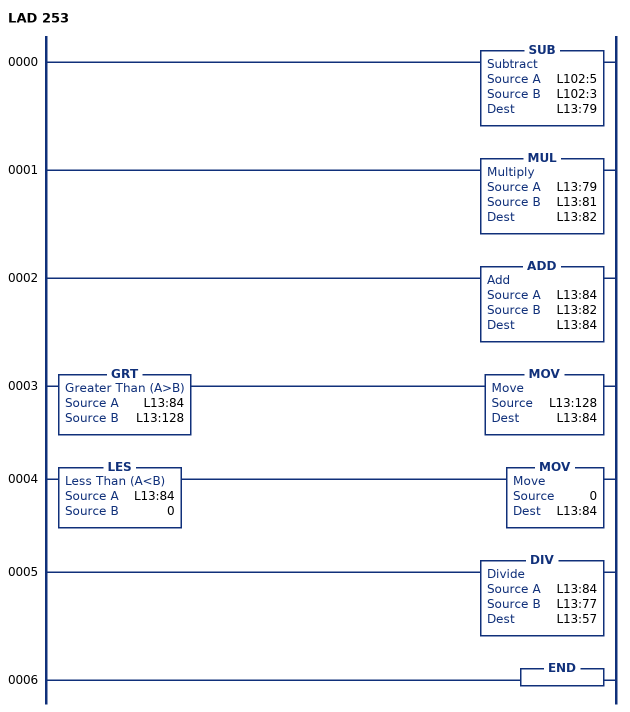
% Rung: 0 %
SOR SUB L102:5 L102:3 L13:79 EOR
% Rung: 1 %
SOR MUL L13:79 L13:81 L13:82 EOR
% Rung: 2 %
SOR ADD L13:84 L13:82 L13:84 EOR
% Rung: 3 %
SOR GRT L13:84 L13:128 MOV L13:128 L13:84 EOR
% Rung: 4 %
SOR LES L13:84 0 MOV 0 L13:84 EOR
% Rung: 5 %
SOR DIV L13:84 L13:77 L13:57 EOR
% Rung: 6 %
SOR END EOR

LADDER 254
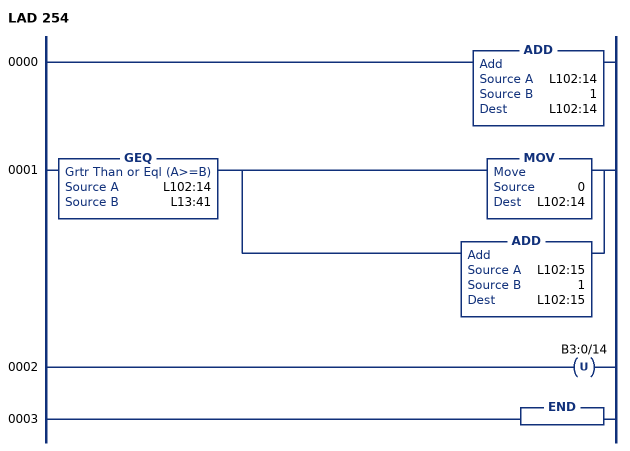
% Rung: 0 %
SOR ADD L102:14 1 L102:14 EOR
% Rung: 1 %
SOR GEQ L102:14 L13:41 BST MOV 0 L102:14 NXB ADD L102:15 1 L102:15 BND EOR
% Rung: 2 %
SOR OTU B3:0/14 EOR
% Rung: 3 %
SOR END EOR

LADDER 255
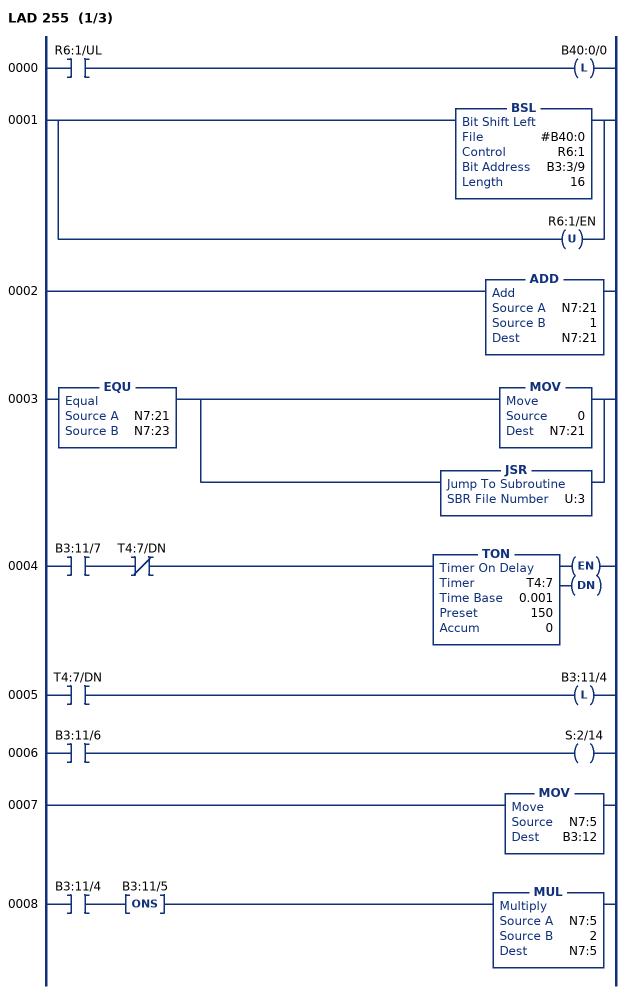
% Rung: 0 %
SOR XIC R6:1/UL OTL B40:0/0 EOR
% Rung: 1 %
SOR BST BSL #B40:0 R6:1 B3:3/9 16 NXB OTU R6:1/EN BND EOR
% Rung: 2 %
SOR ADD N7:21 1 N7:21 EOR
% Rung: 3 %
SOR EQU N7:21 N7:23 BST MOV 0 N7:21 NXB JSR U:3 BND EOR
% Rung: 4 %
SOR XIC B3:11/7 XIO T4:7/DN TON T4:7 0.001 150 0 EOR
% Rung: 5 %
SOR XIC T4:7/DN OTL B3:11/4 EOR
% Rung: 6 %
SOR XIC B3:11/6 OTE S:2/14 EOR
% Rung: 7 %
SOR MOV N7:5 B3:12 EOR
% Rung: 8 %
SOR XIC B3:11/4 ONS B3:11/5 MUL N7:5 2 N7:5 EOR

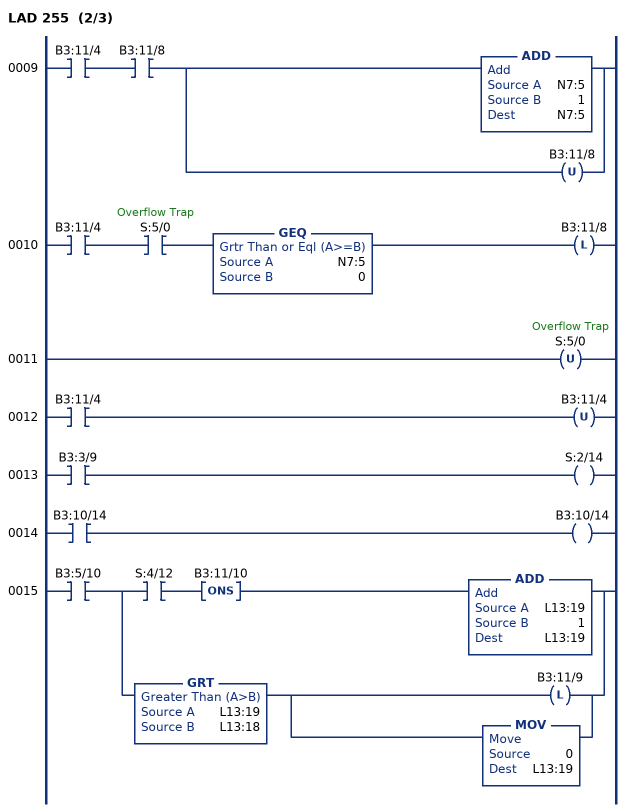
% Rung: 9 %
SOR XIC B3:11/4 XIC B3:11/8 BST ADD N7:5 1 N7:5 NXB OTU B3:11/8 BND EOR
% Rung: 10 %
SOR XIC B3:11/4 XIC S:5/0 GEQ N7:5 0 OTL B3:11/8 EOR
%   S:5/0  "Overflow Trap" %
% Rung: 11 %
SOR OTU S:5/0 EOR
%   S:5/0  "Overflow Trap" %
% Rung: 12 %
SOR XIC B3:11/4 OTU B3:11/4 EOR
% Rung: 13 %
SOR XIC B3:3/9 OTE S:2/14 EOR
% Rung: 14 %
SOR XIC B3:10/14 OTE B3:10/14 EOR
% Rung: 15 %
SOR XIC B3:5/10 BST XIC S:4/12 ONS B3:11/10 ADD L13:19 1 L13:19 NXB GRT L13:19 L13:18 BST OTL B3:11/9 NXB MOV 0 L13:19 BND BND EOR

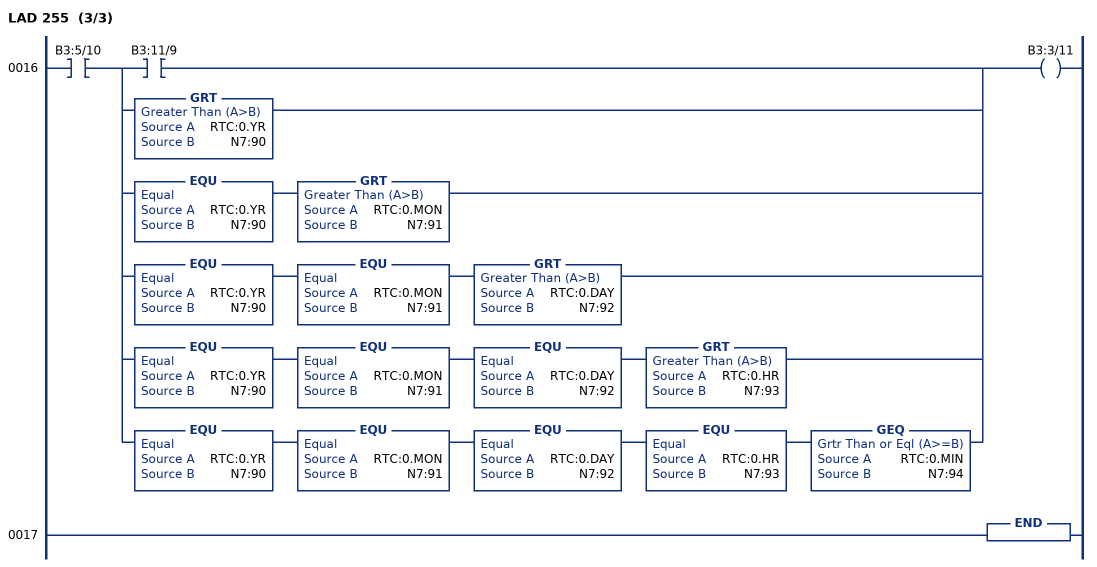
% Rung: 16 %
SOR XIC B3:5/10 BST XIC B3:11/9 NXB GRT RTC:0.YR N7:90 NXB EQU RTC:0.YR N7:90 GRT RTC:0.MON N7:91 NXB EQU RTC:0.YR N7:90 EQU RTC:0.MON N7:91 GRT RTC:0.DAY N7:92 NXB EQU RTC:0.YR N7:90 EQU RTC:0.MON N7:91 EQU RTC:0.DAY N7:92 GRT RTC:0.HR N7:93 NXB EQU RTC:0.YR N7:90 EQU RTC:0.MON N7:91 EQU RTC:0.DAY N7:92 EQU RTC:0.HR N7:93 GEQ RTC:0.MIN N7:94 BND OTE B3:3/11 EOR
% Rung: 17 %
SOR END EOR

DATA TABLE (non-zero values as saved)
DATA B3
% B3:0 % 0X88A2 0X0160 0X0001 0X5101 0X08A5 0X1540 0X0410 0X0461 0X5F80 0X2558
% B3:10 % 0X2000 0X40C7 0X4000 0X08D5 0X0000 0X0000 0X0000 0X0000 0X0000 0X0000
% B3:50 % 0X0001 0X0000 0X0000 0X0000 0X0000 0X0000 0X0000 0X0000 0X0000 0X0000
DATA T4
% .PRE .ACC %
% T4:0 % 0 1
% T4:1 % 150 0
% T4:2 % 400 0
% T4:3 % 222 61
% T4:4 % 1000 0
% T4:5 % 5 5
% T4:6 % 10 32766
% T4:7 % 150 0
% T4:8 % 20 13
% T4:9 % 50 44
% T4:10 % 200 0
% T4:11 % 111 0
% T4:12 % 40 96
% T4:13 % 250 0
% T4:14 % 666 0
% T4:15 % 1000 1006
% T4:16 % 400 0
% T4:17 % 100 96
% T4:18 % 5 0
% T4:19 % 300 0
% T4:20 % 200 0
% T4:21 % 200 0
% T4:22 % 200 0
% T4:23 % 250 0
% T4:24 % 666 0
% T4:25 % 666 0
% T4:26 % 666 0
% T4:27 % 250 0
% T4:28 % 250 0
% T4:29 % 5000 0
% T4:30 % 333 0
% T4:31 % 333 63
% T4:32 % 15 0
% T4:33 % 222 51
% T4:34 % 1111 0
DATA C5
% .PRE .ACC %
% C5:0 % 32766 0
DATA R6
% .LEN .POS %
% R6:0 % 1250 0
% R6:1 % 16 0
% R6:2 % 1050 0
% R6:3 % 1050 0
% R6:4 % 1250 0
% R6:5 % 1250 0
% R6:6 % 1713 0
% R6:7 % 16 0
% R6:8 % 1024 0
% R6:9 % 3 0
% R6:10 % 1713 0
% R6:11 % 1050 0
% R6:12 % 10 0
% R6:13 % 10 0
% R6:14 % 10 0
% R6:15 % 10 0
% R6:16 % 1713 0
% R6:17 % 1713 0
% R6:18 % 1050 0
% R6:19 % 10 0
DATA N7
% N7:0 % 32767 3 874 300 3 0 0 0 500 43
% N7:10 % 1000 43 0 8 8 8 1000 2000 50 1050
% N7:20 % 0 1329 16 2000 0 8 0 0 0 250
% N7:30 % 666 32767 150 0 728 1232 77 32 0 32
% N7:40 % 0 38 1 37 121 482 767 1350 16 0
% N7:50 % 0 0 0 16 1 900 0 0 32766 3
% N7:60 % 1713 1713 1050 871 1034 1024 4999 5 400 400
% N7:70 % 100 200 300 400 90 190 290 390 232 32767
% N7:80 % 0 0 1241 32767 1300 1310 61 26 10 1
% N7:90 % 2011 4 4 12 1 51 25 222 222 12
% N7:100 % 1003 90 110 100 175 25 0 0 0 0
% N7:190 % -128 27477 27605 32767 0 0 0 0 0 0
DATA F8
% F8:0 % 6
DATA L13
% L13:0 % 71471 190025 0 39179 291035
% L13:5 % 6415 33021 6415 172394 5190
% L13:10 % 5004 212369 41937 15 90
% L13:15 % 808527807 -2147483648 2147483647 2147483647 82058
% L13:20 % 147282566 -2001678473 777 36345 100
% L13:25 % 4777 7405 212365 0 713785867
% L13:30 % 94741822 6415 60000 -300674159 1444
% L13:35 % 0 5 99 1073770676 1073770698
% L13:40 % 0 1000000000 1000000 -291038042 -290955777
% L13:45 % 271741302 22 682 26 147282566
% L13:50 % 1099483545 682 1312162756 0 1099483625
% L13:55 % 283196 88766043 1774 47928606 47931497
% L13:60 % 7405 1860375 0 600 -1
% L13:65 % 100 -100 1088103355 -1153047802 1099483566
% L13:70 % 147282479 -1705050752 8 0 147282566
% L13:75 % 0 30 100 -392888222 5
% L13:80 % 40 74 370 40 177378
% L13:85 % 3144934 0 0 0 1099483588
% L13:90 % 283197 3 56648 5 -290955660
% L13:95 % 14 200235 0 271741575 10324515
% L13:100 % 400 7 2147483647 1111 1353
% L13:105 % 10324515 10670 147259324 212376 147259318
% L13:110 % 6 100 50 -2004823403 -2004823412
% L13:115 % -2004823407 5 3 -2004823410 26
% L13:120 % 87 212373 50 100 10
% L13:125 % 0 147282479 2147483647 3276500 3144930
% L13:130 % 2 2 0 99 0
% L13:135 % 0 0 3144930 5 70
% L13:140 % 0 5 36 50 50
% L13:145 % 683 5 88766044 5 0
% L13:150 % 12 20 4 -4 212369
% L13:155 % 0 -10 0 1 4589052
% L13:160 % 12573529 117 273 1220 45
% L13:165 % -2001679672 -2014253201 -2001679672 -2014253201 6706
% L13:170 % 12817 8 225 100 -2147483648
% L13:175 % 4 4 42 23 38
% L13:180 % 1088103355 0 0 1000000 0
% L13:185 % 0 0 -1153047802 0 0
DATA L19
% L19:0 % 713785867 713786507 713796116 713798249 713799019
% L19:5 % 713800070 713825116 713774048 713774596 713774802
% L19:10 % 713777491 713778421 713779204 713779851 713780015
% L19:15 % 713785499 713785672 0 0 0
DATA L20
% L20:0 % -290964835 -290964827 -290964819 -290964811 -290964803
% L20:5 % -290964795 -290964787 -290964779 -290964771 -290964763
% L20:10 % -290964755 -290964747 -290964739 -290964731 -290964723
% L20:15 % -290964715 -290964707 -290964699 -290964691 -290964683
% L20:20 % -290964675 -290964667 -290956009 -290956001 -290955993
% L20:25 % -290955985 -290955977 -290955969 -290955961 -290955953
% L20:30 % -290955945 -290955937 -290955929 -290955921 -290955913
% L20:35 % -290955905 -290955897 -290955889 -290955881 -290955873
% L20:40 % -290955865 -290955857 -290955849 -290955841 -290955833
% L20:45 % -290955825 -290955817 -290955809 -290955801 -290955793
% L20:50 % -290955785 -290955777 -290955769 -290955761 -290955753
% L20:55 % -290955745 -290955737 -290955729 -290955721 -290955713
% L20:60 % -290955705 -290955697 -290990460 -290986195 -290983780
% L20:65 % -290983772 -290983764 -290983756 -290983748 -290983740
% L20:70 % -290983732 -290983724 -290983716 -290981579 -290981571
% L20:75 % -290981563 -290981555 -290981547 -290981539 -290981531
% L20:80 % -290981523 -290981515 -290978966 -290978958 -290978950
% L20:85 % -290978942 -290978934 -290978926 -290978918 -290978910
% L20:90 % -290978902 -290964907 -290964899 -290964891 -290964883
% L20:95 % -290964875 -290964867 -290964859 -290964851 -290964843
DATA L21
% L21:0 % -2001679672 -2001679672 -2001679672 -2001679672 -2001679672
% L21:5 % -2001679672 -2001679672 -2001679672 -2001679672 -2001679672
% L21:10 % -2001679672 -2001679672 -2001679672 -2001679672 -2001679672
% L21:15 % -2001679672 -2001679672 -2001679672 -2001679672 -2001679672
% L21:20 % -2001679672 -2001679672 -2001679672 -2001679672 -2001679672
% L21:25 % -2001679672 -2001679672 -2001679672 -2001679672 -2001679672
% L21:30 % -2001679672 -2001679672 -2001679672 -2001679672 -2001679672
% L21:35 % -2001679672 -2001679672 -2001679672 -2001679672 -2001679672
% L21:40 % -2001679672 -2001679672 -2001679672 -2001679672 -2001679672
% L21:45 % -2001679672 -2001679672 -2001679672 -2001679672 -2001679672
% L21:50 % -2001679672 -2001679672 -2001679672 -2001679672 -2001679672
% L21:55 % -2001679672 -2001679672 -2001679672 -2001679672 -2001679672
% L21:60 % -2001679672 -2001679672 -2001679672 -2001679672 -2001679672
% L21:65 % -2001679672 -2001679672 -2001679672 -2001679672 -2001679672
% L21:70 % -2001679672 -2001679672 -2001679672 -2001679672 -2001679672
% L21:75 % -2001679672 -2001679672 -2001679672 -2001679672 -2001679672
% L21:80 % -2001679672 -2001679672 -2001679672 -2001679672 -2001679672
% L21:85 % -2001679672 -2001679672 -2001679672 -2001679672 -2001679672
% L21:90 % -2001679672 -2001679672 -2001679672 -2001679672 -2001679672
% L21:95 % -2001679672 -2001679672 -2001679672 -2001679672 -2001679672
DATA L22
% L22:0 % 267558685 267558910 267559136 267559362 267559587
% L22:5 % 267559812 267560037 267890042 267890268 267890493
% L22:10 % 267890718 267890944 267891169 267891394 267891619
% L22:15 % 267891844 267892069 271739492 271739718 271739944
% L22:20 % 271740169 271740396 271740622 271740849 271741074
% L22:25 % 271741302 271741527 209710163 209710387 209710612
% L22:30 % 209710838 209711063 209711289 209711514 209711739
% L22:35 % 209711963 209712189 210322365 210322590 210322815
% L22:40 % 210323041 210323267 210323493 210323720 210323946
% L22:45 % 210324172 210324400 267558010 267558235 267558460
DATA L23
% L23:0 % -2014258328 -2014258328 -2014258328 -2014258327 -2014258327
% L23:5 % -2014258327 -2014258327 -2014257928 -2014257927 -2014257927
% L23:10 % -2014257926 -2014257926 -2014257926 -2014257926 -2014257925
% L23:15 % -2014257925 -2014257925 -2014253275 -2014253269 -2014253262
% L23:20 % -2014253254 -2014253245 -2014253235 -2014253224 -2014253213
% L23:25 % -2014253201 -2014253190 -2016530816 -2016530816 -2016530815
% L23:30 % -2016530815 -2016530815 -2016530815 -2016530814 -2016530814
% L23:35 % -2016530813 -2016530813 -2016529979 -2016529927 -2016529864
% L23:40 % -2016529790 -2016529705 -2016529611 -2016529509 -2016529400
% L23:45 % -2016529284 -2016529161 -2014258329 -2014258328 -2014258328
DATA L30
% L30:0 % 124899812 124900038 124900263 124900489 124901389
% L30:5 % 124901614 124901839 124902065 124902967 124903193
% L30:10 % 124903417 124903642 271736154 271739422 271739648
% L30:15 % 271739875 271740101 271740328 271740554 271740780
% L30:20 % 271741005 271741231 271741456 -396657169 -396654322
% L30:25 % -396654096 -396653869 -396653643 -396653417 -396652510
% L30:30 % -396652282 -300674185 -291038042 124892592 124893495
% L30:35 % 124893721 124893946 124894172 124895074 124895299
% L30:40 % 124895524 124895750 124896653 124896879 124897104
% L30:45 % 124897330 124898234 124898459 124898684 124898910
DATA L31
% L31:0 % 138409566 138409658 138409748 138409840 138410203
% L31:5 % 138410293 138410384 138410475 138410839 138410930
% L31:10 % 138411020 138411111 138513980 138513980 138513980
% L31:15 % 138513980 138513980 138513980 138513980 138513980
% L31:20 % 138513980 138513980 138513980 147282566 147282566
% L31:25 % 147282566 147282566 147282566 147282566 147282566
% L31:30 % 147282566 147282566 147282566 138406654 138407018
% L31:35 % 138407109 138407200 138407291 138407655 138407746
% L31:40 % 138407836 138407927 138408292 138408383 138408474
% L31:45 % 138408565 138408929 138409020 138409111 138409202
DATA L32
% L32:0 % -392888994 1309923752 1309923977 1309924203 1309924429
% L32:5 % 1309924654 1309924879 1310035435 1311226092 1312068808
% L32:10 % 1312161404 1312161629 1312161854 1312162079 1312162305
% L32:15 % 1312162530 1312162756 1312162982 1312163207 1312163433
% L32:20 % -1676295510 -1676295285 -1676295060 -1676294835 -1676294609
% L32:25 % -1676294384 -1676294158 -1676293933 -1676293708 -1676293482
% L32:30 % -392891794 1078901975 1078902201 1307407687 1307407912
% L32:35 % 1307408137 1307408362 1307408587 1307408812 1307409037
% L32:40 % 1307409262 1307409488 713775181 713775345 713780829
% L32:45 % 713780999 713781193 713781834 713791450 713793581
DATA L33
% L33:0 % 147282566 146744846 146744846 146744846 146744846
% L33:5 % 146744846 146744846 146747577 147047625 147260001
% L33:10 % 147282285 147282334 147282378 147282418 147282451
% L33:15 % 147282479 147282501 147282520 147282534 147282545
% L33:20 % 147282566 147282566 147282566 147282566 147282566
% L33:25 % 147282566 147282566 147282566 147282566 147282566
% L33:30 % 147282566 146744846 146744846 146744846 146744846
% L33:35 % 146744846 146744846 146744846 146744846 146744846
% L33:40 % 146744846 146744846 146717157 146717202 146718694
% L33:45 % 146718740 146718793 146718967 146721583 146722163
DATA B34
% B34:0 % 0X0000 0X0000 0X0000 0X0000 0X0000 0X0000 0X0000 0X0200 0X0000 0X0000
% B34:40 % 0X0000 0X0000 0X0100 0X2000 0X0100 0X0040 0X0200 0X8000 0X0000 0X0800
% B34:50 % 0X0000 0X1000 0X0000 0X0000 0X0010 0X0000 0X0000 0X0001 0X0000 0X0000
% B34:60 % 0X0002 0X0000 0X0000 0X0000 0X0000 0X0000 0X0000 0X0000 0X0000 0X0000
DATA B35
% B35:110 % 0X0000 0X0000 0X0200 0X0000 0X0000 0X0000 0X0000 0X0000 0X0000 0X0000
DATA B36
% B36:40 % 0X0000 0X0000 0X0000 0X2000 0X0000 0X0000 0X0000 0X0000 0X0000 0X0000
DATA B40
% B40:0 % 0XAAAA
DATA B100
% B100:0 % 0X2700 0X0800 0X0004 0X0000 0X0000 0X0000 0X0000 0X0000 0X0000 0X0000
DATA N101
% N101:0 % 121 682 0 0 1184 100 867 1200 1200 1241
% N101:10 % 1249 1503 10 20642 1269 17365 6 222 333 333
% N101:20 % 1000 500 400 1 0 10 222 15 0 0
DATA L102
% L102:0 % 40 10 1 1 6500
% L102:5 % 6500 0 0 0 0
% L102:10 % 0 1 0 0 56648
% L102:15 % 0 30 10 30 10
% L102:20 % 68744 1 11004 13 117
% L102:25 % 26 0 4 10300330 0
% L102:30 % -1705050752 0 88750944 24170 1587202
% L102:35 % 0 350 1 999999 273
% L102:40 % 0 -668398265 11624 -9544372 0
